FUNCTION_BLOCK FB_PathGenerator
VAR_INPUT
	bStart : BOOL;
	TIN : TIME;
END_VAR
VAR_OUTPUT
	Qout : BOOL; // Finished
	t : LREAL;
END_VAR
VAR
	tTimer : TON;
	tElappsed : TIME;
END_VAR

tTimer(IN := bStart, 
		PT := TIN,
		Q => Qout,
		ET => tElappsed);

t := TIME_TO_LREAL(tElappsed)/1000; // Time to S

END_FUNCTION_BLOCK

(* stored: Version 1.1.0.1, ProductVersion 3.1.4024.12
   POU FB_PathGenerator: Id {c435b4ab-f20b-4b44-b229-cbaec632384b}, SpecialFunc None *)
